KUKA KRL program: check_right_tool.src, check_right_tool.dat

--- check_right_tool.src ---
&ACCESS RVO8
&REL 2
&PARAM TEMPLATE = C:\KRC\Roboter\Template\vorgabe
&PARAM EDITMASK = *
DEF CHECK_RIGHT_TOOL( )

;FOLD ; STATION P13060;%{PE}%R 4.1.16,%MKUKATPBASIS,%CCOMMENT,%VNORMAL,%P 2:STATION P13060
;ENDFOLD
;FOLD ; ROBOT 4;%{PE}%R 4.1.16,%MKUKATPBASIS,%CCOMMENT,%VNORMAL,%P 2:ROBOT 4
;ENDFOLD
;FOLD ; MODULO DE CHECAGEM DA FERRAMENTA;%{PE}%R 4.1.16,%MKUKATPBASIS,%CCOMMENT,%VNORMAL,%P 2:MODULO DE CHECAGEM DA FERRAMENTA
;ENDFOLD

;%%%%%%%%%%%%%%%%% ATENTION %%%%%%%%%%%%%%%%%%%%%
;%%%%%%%% THE GUN USED IT`S NOT CORRECT %%%%%%%%%
;%%% CHECK THE GUN OR THE SIGNAL ON THE DOCK %%%%
;%%%%%%%%%%%% START WITH THE GUN C1 %%%%%%%%%%%%%
;-----------------------------------------------
;%%%%%%%%%%%%%%%%% ATENCAO !!! %%%%%%%%%%%%%%%%%%
;%%% PINCA QUE ESTA SENDO UTILIZADA NO MOMENTO %%
;%%%%%%% NAO E A CORRETA, UTILIZE A GUN C1 %%%%%%
;%%%%%%% OU VERIFIQUE O SINAL DO DOCK %%%%%%%%%%%

WAIT FOR (NOT $IN[169]) AND ($IN[161]) AND ($IN[177]) AND ($IN[219])



END

--- check_right_tool.dat ---
&ACCESS RVO8
&REL 2
&PARAM TEMPLATE = C:\KRC\Roboter\Template\vorgabe
&PARAM EDITMASK = *
DEFDAT CHECK_RIGHT_TOOL
;FOLD EXTERNAL DECLARATIONS;%{PE}%V3.2.0,%MKUKATPBASIS,%CEXT,%VCOMMON,%P
;FOLD BAS EXT;%{PE}%V3.2.0,%MKUKATPBASIS,%CEXT,%VEXT,%P
EXT  BAS (BAS_COMMAND  :IN,REAL  :IN )
DECL INT SUCCESS
;ENDFOLD
;FOLD A10 EXT;%{E}%V3.2.0,%MKUKATPARC,%CEXT,%VEXT,%P
EXT  A10 (A_CMD_T:IN,A_STRT_T:IN,A_WELD_T:IN,A_END_T:IN,INT:IN)
;ENDFOLD
;FOLD A20 EXT;%{E}%V3.2.0,%MKUKATPA20,%CEXT,%VEXT,%P
EXT  A20 (INT  :IN,WELD_ST:IN,WELD_FI:IN,INT:IN)
;ENDFOLD
;FOLD GRIPPER EXT;%{E}%V3.2.0,%MKUKATPGRIPPER,%CEXT,%VEXT,%P
EXT  H50 (INT:IN, INT:IN ,INT:IN ,GRP_TYP:IN)
;ENDFOLD
;FOLD SPOT EXT;%{E}%V3.2.0,%MKUKATPSPOT,%CEXT,%VEXT,%P
EXT  USERSPOT (S_COMMAND  :IN, SPOT_TYPE:IN)
;ENDFOLD
;FOLD TOUCHSENSE EXT;%{E}%V3.2.0,%MKUKATPTS,%CEXT,%VEXT,%P
EXT  H70 (INT  :IN,SRCH_TYP_2  :OUT,E6POS  :IN,SRCH_TYP_3  :IN,SRCH_TYP_2  :IN,SRCH_TYP_2  :IN,SRCH_TYP_2  :IN,SRCH_TYP_2  :IN,SRCH_TYP_2  :IN,INT  :IN )
;ENDFOLD
;FOLD USER EXT;%{E}%V3.2.0,%MKUKATPUSER,%CEXT,%VEXT,%P
;Make here your modifications
;ENDFOLD
;ENDFOLD

ENDDAT
